// TIA Portal V18 export
// export: Created 2026-06-08T16:04:36.8605459Z, ExportSetting WithDefaults, DisplayName Totally Integrated Automation Portal, DisplayVersion V18, DisplayName TIA Portal Openness, DisplayVersion V18, DisplayName TIA Portal Version Control Interface, DisplayVersion V18, DisplayName STEP 7 Professional, DisplayVersion V18, DisplayName STEP 7 Safety, DisplayVersion V18, DisplayName WinCC Professional, DisplayVersion V18
VAR_GLOBAL   // PLC tag table "SO_NGUYEN"
   Act_Count_Cao AT %MW200 : Int;   // Bộ đếm số sản phẩm trọng lượng nhẹ
   Act_Count_TB AT %MW202 : Int;   // Bộ đếm số sản phẩm trọng lượng trung bình
   Act_Count_Thap AT %MW204 : Int;   // Bộ đếm số sản phẩm trọng lượng nặng
   Simu_VT_SP AT %MW206 : Int;   // Mô phỏng vị trí sản phẩm
   Simu_Type_SP AT %MW208 : Int;   // Mô phỏng loại sản phẩm
END_VAR
